FUNCTION_BLOCK FB_TensionLoop
VAR_INPUT
 Enable:			BOOL;
 SetTension:		REAL;
 ActTension:		REAL;
 Hold:				BOOL;
 Invert:			BOOL;
//	stParams:		ST_CTRL_PID_PARAMS;
 Kp:				LREAL;
 Tn:				TIME;
 Td:				TIME;
 PidOutMaxValue:	LREAL;
 PidOutMinValue:	LREAL;	
	
END_VAR
VAR_OUTPUT
	CorrectionSpeed:	REAL;
END_VAR
VAR
 Error:	REAL;
 PID:				FB_CTRL_PID;
 PidLimiter:		FB_CTRL_LIMITER;
 Pidstparams:		ST_CTRL_PID_PARAMS;
 LimiterstParams:	ST_CTRL_LIMITER_PARAMS;	
	
 fbGetCurTaskIdx: 		GETCURTASKINDEX;
 TaskCycleTimeUDINT: 	UDINT;
 TaskCycleTime: 		TIME;
END_VAR


IF (TaskCycleTimeUDINT = 0) THEN
	fbGetCurTaskIdx();
	TaskCycleTimeUDINT := _TaskInfo[fbGetCurTaskIdx.index].CycleTime;
	TaskCycleTime	:= UDINT_TO_TIME(TaskCycleTimeUDINT/10000); 
END_IF


IF (Enable = FALSE) THEN
	pid.eMode	:= eCTRL_MODE_IDLE;
ELSE
	pid.eMode	:= eCTRL_MODE_ACTIVE;	
END_IF

// Call PID function	

PID.fSetpointValue	:= SetTension; 
PID.fActualValue	:= ActTension; 
PID.bHold			:= Hold;

Pidstparams.fKp	:= Kp; 
Pidstparams.tTn	:= Tn; 
Pidstparams.tTd	:= Td; 
Pidstparams.fOutMaxLimit	:= PidOutMaxValue;
Pidstparams.fOutMinLimit	:= PidOutMinValue;
Pidstparams.tCtrlCycleTime	:= TaskCycleTime; 
Pidstparams.tTaskCycleTime	:= TaskCycleTime;

PID(stParams := Pidstparams);

// Call Limiter function

LimiterstParams.tTaskCycleTime	:= TaskCycleTime;
LimiterstParams.tCtrlCycleTime	:= TaskCycleTime;
LimiterstParams.fMaxOutput		:= Pidstparams.fOutMaxLimit;
LimiterstParams.fMinOutput		:= Pidstparams.fOutMinLimit;

PidLimiter.fIn	:= PID.fOut; 
PidLimiter(stParams := LimiterstParams);

IF (Invert = FALSE) THEN
	CorrectionSpeed	:= LREAL_TO_REAL(PidLimiter.fOut);
ELSE
	CorrectionSpeed	:= LREAL_TO_REAL(- PidLimiter.fOut);	
END_IF

END_FUNCTION_BLOCK

(* stored: Version 1.1.0.1, ProductVersion 3.1.4024.3
   POU FB_TensionLoop: Id {6a309c82-5169-0702-0047-e6d555b4cbf9}, SpecialFunc None *)
